{attribute 'conditionalshow'}
PROGRAM INTERNAL PRG_ScopedContextStack
VAR
	aContextStack		: ARRAY[1..SIZEOF(TwinCAT_SystemInfoVarList._TaskInfo)/SIZEOF(PlcTaskSystemInfo)] OF ST_ScopedContextStack;
END_VAR

PROPERTY INTERNAL TaskContextStack : REFERENCE TO ST_ScopedContextStack
GET
VAR
	nTaskIdx	: DINT;
END_VAR
nTaskIdx := Tc2_System.GETCURTASKINDEXEX();
TaskContextStack REF= aContextStack[nTaskIdx];
END_GET
END_PROPERTY

END_PROGRAM

(* stored: Version 1.1.0.1, ProductVersion 3.1.4024.6
   POU PRG_ScopedContextStack: Id {c32a6184-a03b-4217-9b7b-06a1b2e77d20}, SpecialFunc None
   Property TaskContextStack: Id {ce9ae34e-fa10-4f49-a87d-e55aacc3500f}
   Get Get: Id {60fce572-d48b-4c16-83b1-a567999dbd38} *)
